TYPE CyclicAxis_Status_typ :
	STRUCT	
		CyclicPos:	CyclicPos_Status_typ;	
		CyclicVel:	CyclicVel_Status_typ;	
	END_STRUCT
END_TYPE

(* stored: Version 1.1.0.1, ProductVersion 3.1.4024.3
   DUT CyclicAxis_Status_typ: Id {38f42e55-fdbb-0399-2aae-a987c5e791b9} *)
